// TwinCAT 3 PLC project UiBuilder
// ProgramVersion: 3.1.4026.19
// libraries:
//   Base, * (Photara)
//   Discrete, * (Photara)
//   Motion, * (Photara)
//   Nemo, * (Photara)
//   Tc2_EthernetIP, * (Beckhoff Automation GmbH)
//   Tc2_ProfinetDiag, * (Beckhoff Automation GmbH)
//   Tc2_Standard, * (Beckhoff Automation GmbH)
//   Tc2_System, * (Beckhoff Automation GmbH)
//   Vision, * (Photara)
//   TcUnit, * (www.tcunit.org)
// project tree:
//   DUTs/ ST_HMICommand.TcDUT, ST_HMIConfiguration.TcDUT, ST_HMIComponentAPI.TcDUT, ST_HMIStatus.TcDUT
//   ITFs/ I_HMIBase.TcIO
//   / PlcTask.TcTTO
//   POUs/ FB_HMIBase.TcPOU, MAIN.TcPOU
//   Tests/ FB_ST_HMICommand_Test.TcPOU, FB_ST_HMIComponentAPI_Test.TcPOU, FB_ST_HMIStatus_Test.TcPOU, FB_HMIBase_Test.TcPOU, PRG_TEST.TcPOU

CONFIGURATION UiBuilder
    RESOURCE PLC ON TwinCAT3
        TASK PlcTask(INTERVAL := T#10ms, PRIORITY := 20);
        PROGRAM MAIN WITH PlcTask : MAIN;
    END_RESOURCE
END_CONFIGURATION

// ---- DUTs/ST_HMICommand.TcDUT
TYPE ST_HMICommand :
STRUCT
	Enable	: BOOL;
	Disable	: BOOL;
	Home	: BOOL;
	Reset	: BOOL;
	Stop	: BOOL;
	Trigger	: BOOL;
	Error	: BYTE;
END_STRUCT
END_TYPE

// ---- DUTs/ST_HMIConfiguration.TcDUT
TYPE ST_HMIConfiguration :
STRUCT
	ComponentConfiguration : REFERENCE TO ST_CommandConfiguration;
END_STRUCT
END_TYPE

// ---- DUTs/ST_HMIComponentAPI.TcDUT
TYPE ST_HMIComponentAPI :
STRUCT 
	Done : BOOL;
	Busy : BOOL;
	Error : BOOL;
	ErrorID : BOOL;
	Ready : BOOL;
	Enabled: BOOL;
	Homed: BOOL;
	Moving : BOOL;
END_STRUCT
END_TYPE

// ---- DUTs/ST_HMIStatus.TcDUT
TYPE ST_HMIStatus :
STRUCT
	ComponentStatus : REFERENCE TO ST_ComponentStatus;
	HmiStatus : ST_HmiComponentAPI;
END_STRUCT
END_TYPE

// ---- ITFs/I_HMIBase.TcIO
INTERFACE I_HMIBase EXTENDS	Base.I_BaseCyclic

PROPERTY P_BaseConfiguration : REFERENCE TO ST_BaseConfiguration
GET
END_GET
SET
END_SET
END_PROPERTY

PROPERTY P_BaseStatus : REFERENCE TO ST_BaseStatus
GET
END_GET
SET
END_SET
END_PROPERTY

PROPERTY P_Command : REFERENCE TO P_Command
GET
END_GET
SET
END_SET
END_PROPERTY

END_INTERFACE

// ---- POUs/MAIN.TcPOU
PROGRAM MAIN
VAR
END_VAR

END_PROGRAM

// ---- POUs/FB_HMIBase.TcPOU
FUNCTION_BLOCK FB_HMIBase
VAR
	status : ST_HMIStatus;
	configs : ST_HMIConfiguration;
	cmd : ST_HMICommand;
END_VAR

PROPERTY P_Command : ST_HMICommand
GET
END_GET
SET
END_SET
END_PROPERTY

PROPERTY P_Configuration : ST_HMIConfiguration
GET
END_GET
SET
END_SET
END_PROPERTY

PROPERTY P_Status : ST_HMIStatus
GET
END_GET
SET
END_SET
END_PROPERTY

END_FUNCTION_BLOCK

// ---- Tests/FB_ST_HMICommand_Test.TcPOU
FUNCTION_BLOCK FB_ST_HMICommand_Test EXTENDS TcUnit.FB_TestSuite
VAR_INPUT
END_VAR
VAR_OUTPUT
END_VAR
VAR
	testCommand : ST_HMICommand;
END_VAR

// Test runner - call all test methods
Test_InitialState();
Test_EnableCommand();
Test_DisableCommand();
Test_HomeCommand();
Test_ResetCommand();
Test_StopCommand();
Test_TriggerCommand();
Test_ErrorCode();
Test_MultipleCommands();
Test_ClearCommands();

METHOD Test_InitialState
VAR_INPUT
END_VAR
TEST('Test_InitialState');

// Test that all command flags are initially FALSE
testCommand.Enable := FALSE;
testCommand.Disable := FALSE;
testCommand.Home := FALSE;
testCommand.Reset := FALSE;
testCommand.Stop := FALSE;
testCommand.Trigger := FALSE;
testCommand.Error := 0;

AssertFalse(testCommand.Enable, 'Enable should be FALSE initially');
AssertFalse(testCommand.Disable, 'Disable should be FALSE initially');
AssertFalse(testCommand.Home, 'Home should be FALSE initially');
AssertFalse(testCommand.Reset, 'Reset should be FALSE initially');
AssertFalse(testCommand.Stop, 'Stop should be FALSE initially');
AssertFalse(testCommand.Trigger, 'Trigger should be FALSE initially');
AssertEquals_BYTE(0, testCommand.Error, 'Error should be 0 initially');

TEST_FINISHED();
END_METHOD

METHOD Test_EnableCommand
VAR_INPUT
END_VAR
TEST('Test_EnableCommand');

// Test Enable command can be set
testCommand.Enable := TRUE;
AssertTrue(testCommand.Enable, 'Enable should be TRUE when set');

// Reset
testCommand.Enable := FALSE;
AssertFalse(testCommand.Enable, 'Enable should be FALSE when reset');

TEST_FINISHED();
END_METHOD

METHOD Test_DisableCommand
VAR_INPUT
END_VAR
TEST('Test_DisableCommand');

// Test Disable command can be set
testCommand.Disable := TRUE;
AssertTrue(testCommand.Disable, 'Disable should be TRUE when set');

// Reset
testCommand.Disable := FALSE;
AssertFalse(testCommand.Disable, 'Disable should be FALSE when reset');

TEST_FINISHED();
END_METHOD

METHOD Test_HomeCommand
VAR_INPUT
END_VAR
TEST('Test_HomeCommand');

// Test Home command can be set
testCommand.Home := TRUE;
AssertTrue(testCommand.Home, 'Home should be TRUE when set');

// Reset
testCommand.Home := FALSE;
AssertFalse(testCommand.Home, 'Home should be FALSE when reset');

TEST_FINISHED();
END_METHOD

METHOD Test_ResetCommand
VAR_INPUT
END_VAR
TEST('Test_ResetCommand');

// Test Reset command can be set
testCommand.Reset := TRUE;
AssertTrue(testCommand.Reset, 'Reset should be TRUE when set');

// Reset
testCommand.Reset := FALSE;
AssertFalse(testCommand.Reset, 'Reset should be FALSE when reset');

TEST_FINISHED();
END_METHOD

METHOD Test_StopCommand
VAR_INPUT
END_VAR
TEST('Test_StopCommand');

// Test Stop command can be set
testCommand.Stop := TRUE;
AssertTrue(testCommand.Stop, 'Stop should be TRUE when set');

// Reset
testCommand.Stop := FALSE;
AssertFalse(testCommand.Stop, 'Stop should be FALSE when reset');

TEST_FINISHED();
END_METHOD

METHOD Test_TriggerCommand
VAR_INPUT
END_VAR
TEST('Test_TriggerCommand');

// Test Trigger command can be set
testCommand.Trigger := TRUE;
AssertTrue(testCommand.Trigger, 'Trigger should be TRUE when set');

// Reset
testCommand.Trigger := FALSE;
AssertFalse(testCommand.Trigger, 'Trigger should be FALSE when reset');

TEST_FINISHED();
END_METHOD

METHOD Test_ErrorCode
VAR_INPUT
END_VAR
TEST('Test_ErrorCode');

// Test Error code can be set to various values
testCommand.Error := 0;
AssertEquals_BYTE(0, testCommand.Error, 'Error should be 0');

testCommand.Error := 1;
AssertEquals_BYTE(1, testCommand.Error, 'Error should be 1');

testCommand.Error := 255;
AssertEquals_BYTE(255, testCommand.Error, 'Error should be 255');

testCommand.Error := 128;
AssertEquals_BYTE(128, testCommand.Error, 'Error should be 128');

TEST_FINISHED();
END_METHOD

METHOD Test_MultipleCommands
VAR_INPUT
END_VAR
TEST('Test_MultipleCommands');

// Test multiple commands can be set simultaneously
testCommand.Enable := TRUE;
testCommand.Home := TRUE;
testCommand.Trigger := TRUE;

AssertTrue(testCommand.Enable, 'Enable should be TRUE');
AssertTrue(testCommand.Home, 'Home should be TRUE');
AssertTrue(testCommand.Trigger, 'Trigger should be TRUE');
AssertFalse(testCommand.Disable, 'Disable should remain FALSE');
AssertFalse(testCommand.Stop, 'Stop should remain FALSE');

TEST_FINISHED();
END_METHOD

METHOD Test_ClearCommands
VAR_INPUT
END_VAR
TEST('Test_ClearCommands');

// Set all commands
testCommand.Enable := TRUE;
testCommand.Disable := TRUE;
testCommand.Home := TRUE;
testCommand.Reset := TRUE;
testCommand.Stop := TRUE;
testCommand.Trigger := TRUE;
testCommand.Error := 42;

// Clear all commands
testCommand.Enable := FALSE;
testCommand.Disable := FALSE;
testCommand.Home := FALSE;
testCommand.Reset := FALSE;
testCommand.Stop := FALSE;
testCommand.Trigger := FALSE;
testCommand.Error := 0;

// Verify all are cleared
AssertFalse(testCommand.Enable, 'Enable should be FALSE');
AssertFalse(testCommand.Disable, 'Disable should be FALSE');
AssertFalse(testCommand.Home, 'Home should be FALSE');
AssertFalse(testCommand.Reset, 'Reset should be FALSE');
AssertFalse(testCommand.Stop, 'Stop should be FALSE');
AssertFalse(testCommand.Trigger, 'Trigger should be FALSE');
AssertEquals_BYTE(0, testCommand.Error, 'Error should be 0');

TEST_FINISHED();
END_METHOD

END_FUNCTION_BLOCK

// ---- Tests/FB_ST_HMIComponentAPI_Test.TcPOU
FUNCTION_BLOCK FB_ST_HMIComponentAPI_Test EXTENDS TcUnit.FB_TestSuite
VAR_INPUT
END_VAR
VAR_OUTPUT
END_VAR
VAR
	testAPI : ST_HMIComponentAPI;
END_VAR

// Test runner - call all test methods
Test_InitialState();
Test_DoneFlag();
Test_BusyFlag();
Test_ErrorFlag();
Test_ErrorIDFlag();
Test_ReadyFlag();
Test_EnabledFlag();
Test_HomedFlag();
Test_MovingFlag();
Test_StateTransitions();
Test_ErrorState();
Test_BusyToDone();
Test_AllFlagsSet();
Test_ClearAllFlags();

METHOD Test_InitialState
VAR_INPUT
END_VAR
TEST('Test_InitialState');

// Initialize all flags to FALSE
testAPI.Done := FALSE;
testAPI.Busy := FALSE;
testAPI.Error := FALSE;
testAPI.ErrorID := FALSE;
testAPI.Ready := FALSE;
testAPI.Enabled := FALSE;
testAPI.Homed := FALSE;
testAPI.Moving := FALSE;

// Verify initial state
AssertFalse(testAPI.Done, 'Done should be FALSE initially');
AssertFalse(testAPI.Busy, 'Busy should be FALSE initially');
AssertFalse(testAPI.Error, 'Error should be FALSE initially');
AssertFalse(testAPI.ErrorID, 'ErrorID should be FALSE initially');
AssertFalse(testAPI.Ready, 'Ready should be FALSE initially');
AssertFalse(testAPI.Enabled, 'Enabled should be FALSE initially');
AssertFalse(testAPI.Homed, 'Homed should be FALSE initially');
AssertFalse(testAPI.Moving, 'Moving should be FALSE initially');

TEST_FINISHED();
END_METHOD

METHOD Test_DoneFlag
VAR_INPUT
END_VAR
TEST('Test_DoneFlag');

// Test Done flag can be set
testAPI.Done := TRUE;
AssertTrue(testAPI.Done, 'Done should be TRUE when set');

// Reset
testAPI.Done := FALSE;
AssertFalse(testAPI.Done, 'Done should be FALSE when reset');

TEST_FINISHED();
END_METHOD

METHOD Test_BusyFlag
VAR_INPUT
END_VAR
TEST('Test_BusyFlag');

// Test Busy flag can be set
testAPI.Busy := TRUE;
AssertTrue(testAPI.Busy, 'Busy should be TRUE when set');

// Reset
testAPI.Busy := FALSE;
AssertFalse(testAPI.Busy, 'Busy should be FALSE when reset');

TEST_FINISHED();
END_METHOD

METHOD Test_ErrorFlag
VAR_INPUT
END_VAR
TEST('Test_ErrorFlag');

// Test Error flag can be set
testAPI.Error := TRUE;
AssertTrue(testAPI.Error, 'Error should be TRUE when set');

// Reset
testAPI.Error := FALSE;
AssertFalse(testAPI.Error, 'Error should be FALSE when reset');

TEST_FINISHED();
END_METHOD

METHOD Test_ErrorIDFlag
VAR_INPUT
END_VAR
TEST('Test_ErrorIDFlag');

// Test ErrorID flag can be set
testAPI.ErrorID := TRUE;
AssertTrue(testAPI.ErrorID, 'ErrorID should be TRUE when set');

// Reset
testAPI.ErrorID := FALSE;
AssertFalse(testAPI.ErrorID, 'ErrorID should be FALSE when reset');

TEST_FINISHED();
END_METHOD

METHOD Test_ReadyFlag
VAR_INPUT
END_VAR
TEST('Test_ReadyFlag');

// Test Ready flag can be set
testAPI.Ready := TRUE;
AssertTrue(testAPI.Ready, 'Ready should be TRUE when set');

// Reset
testAPI.Ready := FALSE;
AssertFalse(testAPI.Ready, 'Ready should be FALSE when reset');

TEST_FINISHED();
END_METHOD

METHOD Test_EnabledFlag
VAR_INPUT
END_VAR
TEST('Test_EnabledFlag');

// Test Enabled flag can be set
testAPI.Enabled := TRUE;
AssertTrue(testAPI.Enabled, 'Enabled should be TRUE when set');

// Reset
testAPI.Enabled := FALSE;
AssertFalse(testAPI.Enabled, 'Enabled should be FALSE when reset');

TEST_FINISHED();
END_METHOD

METHOD Test_HomedFlag
VAR_INPUT
END_VAR
TEST('Test_HomedFlag');

// Test Homed flag can be set
testAPI.Homed := TRUE;
AssertTrue(testAPI.Homed, 'Homed should be TRUE when set');

// Reset
testAPI.Homed := FALSE;
AssertFalse(testAPI.Homed, 'Homed should be FALSE when reset');

TEST_FINISHED();
END_METHOD

METHOD Test_MovingFlag
VAR_INPUT
END_VAR
TEST('Test_MovingFlag');

// Test Moving flag can be set
testAPI.Moving := TRUE;
AssertTrue(testAPI.Moving, 'Moving should be TRUE when set');

// Reset
testAPI.Moving := FALSE;
AssertFalse(testAPI.Moving, 'Moving should be FALSE when reset');

TEST_FINISHED();
END_METHOD

METHOD Test_StateTransitions
VAR_INPUT
END_VAR
TEST('Test_StateTransitions');

// Simulate typical state transition: Ready -> Busy -> Done
testAPI.Ready := TRUE;
AssertTrue(testAPI.Ready, 'Should be Ready initially');
AssertFalse(testAPI.Busy, 'Should not be Busy initially');
AssertFalse(testAPI.Done, 'Should not be Done initially');

// Transition to Busy
testAPI.Busy := TRUE;
testAPI.Ready := FALSE;
AssertFalse(testAPI.Ready, 'Should not be Ready when Busy');
AssertTrue(testAPI.Busy, 'Should be Busy');
AssertFalse(testAPI.Done, 'Should not be Done while Busy');

// Transition to Done
testAPI.Done := TRUE;
testAPI.Busy := FALSE;
AssertFalse(testAPI.Busy, 'Should not be Busy when Done');
AssertTrue(testAPI.Done, 'Should be Done');

TEST_FINISHED();
END_METHOD

METHOD Test_ErrorState
VAR_INPUT
END_VAR
TEST('Test_ErrorState');

// Simulate error condition
testAPI.Error := TRUE;
testAPI.ErrorID := TRUE;
testAPI.Busy := FALSE;
testAPI.Done := FALSE;

AssertTrue(testAPI.Error, 'Error should be TRUE');
AssertTrue(testAPI.ErrorID, 'ErrorID should be TRUE');
AssertFalse(testAPI.Done, 'Done should be FALSE in error state');
AssertFalse(testAPI.Busy, 'Busy should be FALSE in error state');

TEST_FINISHED();
END_METHOD

METHOD Test_BusyToDone
VAR_INPUT
END_VAR
TEST('Test_BusyToDone');

// Test transition from Busy to Done (should be mutually exclusive)
testAPI.Busy := TRUE;
testAPI.Done := FALSE;
AssertTrue(testAPI.Busy, 'Should be Busy');
AssertFalse(testAPI.Done, 'Done should be FALSE when Busy');

// Complete operation
testAPI.Busy := FALSE;
testAPI.Done := TRUE;
AssertFalse(testAPI.Busy, 'Busy should be FALSE when Done');
AssertTrue(testAPI.Done, 'Should be Done');

TEST_FINISHED();
END_METHOD

METHOD Test_AllFlagsSet
VAR_INPUT
END_VAR
TEST('Test_AllFlagsSet');

// Test that all flags can be set simultaneously (though not typical in practice)
testAPI.Done := TRUE;
testAPI.Busy := TRUE;
testAPI.Error := TRUE;
testAPI.ErrorID := TRUE;
testAPI.Ready := TRUE;
testAPI.Enabled := TRUE;
testAPI.Homed := TRUE;
testAPI.Moving := TRUE;

AssertTrue(testAPI.Done, 'Done should be TRUE');
AssertTrue(testAPI.Busy, 'Busy should be TRUE');
AssertTrue(testAPI.Error, 'Error should be TRUE');
AssertTrue(testAPI.ErrorID, 'ErrorID should be TRUE');
AssertTrue(testAPI.Ready, 'Ready should be TRUE');
AssertTrue(testAPI.Enabled, 'Enabled should be TRUE');
AssertTrue(testAPI.Homed, 'Homed should be TRUE');
AssertTrue(testAPI.Moving, 'Moving should be TRUE');

TEST_FINISHED();
END_METHOD

METHOD Test_ClearAllFlags
VAR_INPUT
END_VAR
TEST('Test_ClearAllFlags');

// Set all flags
testAPI.Done := TRUE;
testAPI.Busy := TRUE;
testAPI.Error := TRUE;
testAPI.ErrorID := TRUE;
testAPI.Ready := TRUE;
testAPI.Enabled := TRUE;
testAPI.Homed := TRUE;
testAPI.Moving := TRUE;

// Clear all flags
testAPI.Done := FALSE;
testAPI.Busy := FALSE;
testAPI.Error := FALSE;
testAPI.ErrorID := FALSE;
testAPI.Ready := FALSE;
testAPI.Enabled := FALSE;
testAPI.Homed := FALSE;
testAPI.Moving := FALSE;

// Verify all are cleared
AssertFalse(testAPI.Done, 'Done should be FALSE');
AssertFalse(testAPI.Busy, 'Busy should be FALSE');
AssertFalse(testAPI.Error, 'Error should be FALSE');
AssertFalse(testAPI.ErrorID, 'ErrorID should be FALSE');
AssertFalse(testAPI.Ready, 'Ready should be FALSE');
AssertFalse(testAPI.Enabled, 'Enabled should be FALSE');
AssertFalse(testAPI.Homed, 'Homed should be FALSE');
AssertFalse(testAPI.Moving, 'Moving should be FALSE');

TEST_FINISHED();
END_METHOD

END_FUNCTION_BLOCK

// ---- Tests/FB_ST_HMIStatus_Test.TcPOU
FUNCTION_BLOCK FB_ST_HMIStatus_Test EXTENDS TcUnit.FB_TestSuite
VAR_INPUT
END_VAR
VAR_OUTPUT
END_VAR
VAR
	testStatus : ST_HMIStatus;
END_VAR

// Test runner - call all test methods
Test_InitialState();
Test_HmiStatusAccess();
Test_HmiStatusFlags();
Test_HmiStatusStateTransitions();

METHOD Test_InitialState
VAR_INPUT
END_VAR
TEST('Test_InitialState');

// Initialize HmiStatus structure
testStatus.HmiStatus.Done := FALSE;
testStatus.HmiStatus.Busy := FALSE;
testStatus.HmiStatus.Error := FALSE;
testStatus.HmiStatus.ErrorID := FALSE;
testStatus.HmiStatus.Ready := FALSE;
testStatus.HmiStatus.Enabled := FALSE;
testStatus.HmiStatus.Homed := FALSE;
testStatus.HmiStatus.Moving := FALSE;

// Verify initial state of HmiStatus member
AssertFalse(testStatus.HmiStatus.Done, 'HmiStatus.Done should be FALSE initially');
AssertFalse(testStatus.HmiStatus.Busy, 'HmiStatus.Busy should be FALSE initially');
AssertFalse(testStatus.HmiStatus.Error, 'HmiStatus.Error should be FALSE initially');
AssertFalse(testStatus.HmiStatus.ErrorID, 'HmiStatus.ErrorID should be FALSE initially');
AssertFalse(testStatus.HmiStatus.Ready, 'HmiStatus.Ready should be FALSE initially');
AssertFalse(testStatus.HmiStatus.Enabled, 'HmiStatus.Enabled should be FALSE initially');
AssertFalse(testStatus.HmiStatus.Homed, 'HmiStatus.Homed should be FALSE initially');
AssertFalse(testStatus.HmiStatus.Moving, 'HmiStatus.Moving should be FALSE initially');

TEST_FINISHED();
END_METHOD

METHOD Test_HmiStatusAccess
VAR_INPUT
END_VAR
TEST('Test_HmiStatusAccess');

// Test that HmiStatus member can be accessed and modified
testStatus.HmiStatus.Ready := TRUE;
AssertTrue(testStatus.HmiStatus.Ready, 'HmiStatus.Ready should be accessible and settable');

testStatus.HmiStatus.Enabled := TRUE;
AssertTrue(testStatus.HmiStatus.Enabled, 'HmiStatus.Enabled should be accessible and settable');

testStatus.HmiStatus.Homed := TRUE;
AssertTrue(testStatus.HmiStatus.Homed, 'HmiStatus.Homed should be accessible and settable');

TEST_FINISHED();
END_METHOD

METHOD Test_HmiStatusFlags
VAR_INPUT
END_VAR
TEST('Test_HmiStatusFlags');

// Test all HmiStatus flags can be set independently
testStatus.HmiStatus.Done := TRUE;
testStatus.HmiStatus.Busy := FALSE;
testStatus.HmiStatus.Error := FALSE;

AssertTrue(testStatus.HmiStatus.Done, 'Done flag should be TRUE');
AssertFalse(testStatus.HmiStatus.Busy, 'Busy flag should be FALSE');
AssertFalse(testStatus.HmiStatus.Error, 'Error flag should be FALSE');

// Change state
testStatus.HmiStatus.Done := FALSE;
testStatus.HmiStatus.Busy := TRUE;

AssertFalse(testStatus.HmiStatus.Done, 'Done flag should be FALSE');
AssertTrue(testStatus.HmiStatus.Busy, 'Busy flag should be TRUE');

TEST_FINISHED();
END_METHOD

METHOD Test_HmiStatusStateTransitions
VAR_INPUT
END_VAR
TEST('Test_HmiStatusStateTransitions');

// Test typical state machine transitions through HmiStatus
// Initial state: Ready
testStatus.HmiStatus.Ready := TRUE;
testStatus.HmiStatus.Enabled := FALSE;
testStatus.HmiStatus.Busy := FALSE;
testStatus.HmiStatus.Done := FALSE;

AssertTrue(testStatus.HmiStatus.Ready, 'Should be Ready initially');

// Enabled state
testStatus.HmiStatus.Enabled := TRUE;
AssertTrue(testStatus.HmiStatus.Enabled, 'Should be Enabled');
AssertTrue(testStatus.HmiStatus.Ready, 'Should remain Ready when Enabled');

// Busy executing
testStatus.HmiStatus.Busy := TRUE;
testStatus.HmiStatus.Done := FALSE;
AssertTrue(testStatus.HmiStatus.Busy, 'Should be Busy');
AssertFalse(testStatus.HmiStatus.Done, 'Should not be Done while Busy');

// Completed
testStatus.HmiStatus.Busy := FALSE;
testStatus.HmiStatus.Done := TRUE;
AssertFalse(testStatus.HmiStatus.Busy, 'Should not be Busy when Done');
AssertTrue(testStatus.HmiStatus.Done, 'Should be Done');

TEST_FINISHED();
END_METHOD

END_FUNCTION_BLOCK

// ---- Tests/FB_HMIBase_Test.TcPOU
FUNCTION_BLOCK FB_HMIBase_Test EXTENDS TcUnit.FB_TestSuite
VAR_INPUT
END_VAR
VAR_OUTPUT
END_VAR
VAR
	testFB : FB_HMIBase;
	testCommand : ST_HMICommand;
	testConfig : ST_HMIConfiguration;
	testStatus : ST_HMIStatus;
END_VAR

// Test runner - call all test methods
Test_FunctionBlockInstantiation();
Test_CommandProperty();how 
Test_ConfigurationProperty();
Test_StatusProperty();
Test_CommandPropertyReadWrite();
Test_StatusPropertyRead();
Test_ConfigurationPropertyReadWrite();

METHOD Test_CommandProperty
VAR_INPUT
END_VAR
VAR
	retrievedCommand : ST_HMICommand;
END_VAR
TEST('Test_CommandProperty');

// Test P_Command property
// Note: This test assumes property implementation will be added
// Once properties are implemented, this will verify getter/setter behavior

// Set up test command
testCommand.Enable := TRUE;
testCommand.Home := TRUE;
testCommand.Reset := FALSE;

// Note: When properties are implemented, uncomment:
// testFB.P_Command := testCommand;
// retrievedCommand := testFB.P_Command;
// AssertTrue(retrievedCommand.Enable, 'Command.Enable should be TRUE');
// AssertTrue(retrievedCommand.Home, 'Command.Home should be TRUE');
// AssertFalse(retrievedCommand.Reset, 'Command.Reset should be FALSE');

// For now, just verify the structure works
AssertTrue(testCommand.Enable, 'Test command Enable flag works');

TEST_FINISHED();
END_METHOD

METHOD Test_CommandPropertyReadWrite
VAR_INPUT
END_VAR
VAR
	writeCommand : ST_HMICommand;
	readCommand : ST_HMICommand;
END_VAR
TEST('Test_CommandPropertyReadWrite');

// Prepare test data
writeCommand.Enable := TRUE;
writeCommand.Disable := FALSE;
writeCommand.Home := TRUE;
writeCommand.Reset := FALSE;
writeCommand.Stop := FALSE;
writeCommand.Trigger := TRUE;
writeCommand.Error := 42;

// When property implementation is complete, this will test:
// 1. Write via property setter
// testFB.P_Command := writeCommand;

// 2. Read via property getter
// readCommand := testFB.P_Command;

// 3. Verify data integrity
// AssertTrue(readCommand.Enable, 'Enable should match written value');
// AssertFalse(readCommand.Disable, 'Disable should match written value');
// AssertTrue(readCommand.Home, 'Home should match written value');
// AssertTrue(readCommand.Trigger, 'Trigger should match written value');
// AssertEquals_BYTE(42, readCommand.Error, 'Error code should match written value');

// Placeholder verification
AssertTrue(writeCommand.Enable, 'Write command prepared correctly');

TEST_FINISHED();
END_METHOD

METHOD Test_ConfigurationProperty
VAR_INPUT
END_VAR
VAR
	retrievedConfig : ST_HMIConfiguration;
END_VAR
TEST('Test_ConfigurationProperty');

// Test P_Configuration property
// Note: This test assumes property implementation will be added

// Set up test configuration
// testConfig is ready to use once properties are implemented

// Note: When properties are implemented, uncomment:
// testFB.P_Configuration := testConfig;
// retrievedConfig := testFB.P_Configuration;

// For now, verify the structure exists
AssertTrue(TRUE, 'Configuration structure is defined');

TEST_FINISHED();
END_METHOD

METHOD Test_ConfigurationPropertyReadWrite
VAR_INPUT
END_VAR
VAR
	writeConfig : ST_HMIConfiguration;
	readConfig : ST_HMIConfiguration;
END_VAR
TEST('Test_ConfigurationPropertyReadWrite');

// Test configuration property read/write
// Configurations are typically set once and read multiple times

// When property implementation is complete:
// testFB.P_Configuration := writeConfig;
// readConfig := testFB.P_Configuration;

// Verify configuration was stored correctly
// (Will need actual configuration values once ST_CommandConfiguration is defined)

// Placeholder verification
AssertTrue(TRUE, 'Configuration property structure is ready for implementation');

TEST_FINISHED();
END_METHOD

METHOD Test_FunctionBlockInstantiation
VAR_INPUT
END_VAR
TEST('Test_FunctionBlockInstantiation');

// Test that FB_HMIBase can be instantiated
// The mere fact that testFB exists and this test runs proves instantiation works
AssertTrue(TRUE, 'FB_HMIBase should be instantiable');

TEST_FINISHED();
END_METHOD

METHOD Test_StatusProperty
VAR_INPUT
END_VAR
VAR
	retrievedStatus : ST_HMIStatus;
END_VAR
TEST('Test_StatusProperty');

// Test P_Status property
// Note: This test assumes property implementation will be added

// Set up test status
testStatus.HmiStatus.Ready := TRUE;
testStatus.HmiStatus.Enabled := TRUE;

// Note: When properties are implemented, uncomment:
// testFB.P_Status := testStatus;
// retrievedStatus := testFB.P_Status;
// AssertTrue(retrievedStatus.HmiStatus.Ready, 'Status.HmiStatus.Ready should be TRUE');
// AssertTrue(retrievedStatus.HmiStatus.Enabled, 'Status.HmiStatus.Enabled should be TRUE');

// For now, verify the structure works
AssertTrue(testStatus.HmiStatus.Ready, 'Test status Ready flag works');

TEST_FINISHED();
END_METHOD

METHOD Test_StatusPropertyRead
VAR_INPUT
END_VAR
VAR
	readStatus : ST_HMIStatus;
END_VAR
TEST('Test_StatusPropertyRead');

// Typically status is read-only from external perspective
// This test verifies status can be read via property

// When property implementation is complete:
// readStatus := testFB.P_Status;

// Verify status flags can be read
// AssertFalse(readStatus.HmiStatus.Error, 'Should be able to read Error flag');
// AssertFalse(readStatus.HmiStatus.Busy, 'Should be able to read Busy flag');

// Placeholder verification
AssertTrue(TRUE, 'Status property structure is ready for implementation');

TEST_FINISHED();
END_METHOD

END_FUNCTION_BLOCK

// ---- Tests/PRG_TEST.TcPOU
PROGRAM PRG_TEST
VAR
	// Test suite instances
	fbCommandTest : FB_ST_HMICommand_Test;
	fbComponentAPITest : FB_ST_HMIComponentAPI_Test;
	fbStatusTest : FB_ST_HMIStatus_Test;
	fbHMIBaseTest : FB_HMIBase_Test;
END_VAR

// ============================================================================
// UiBuilder Library Test Suite
// ============================================================================
// This program runs all unit tests for the UiBuilder library using TcUnit
// framework. Call this program from your main task to execute tests.
//
// Test Coverage:
// - ST_HMICommand data type tests
// - ST_HMIComponentAPI data type tests
// - ST_HMIStatus data type tests
// - FB_HMIBase function block tests
//
// Usage:
// 1. Add PRG_TEST to your PlcTask or call from MAIN
// 2. Build and download the project
// 3. Run the PLC
// 4. Check TcUnit results in the output window
// ============================================================================

// Execute all test suites
// TcUnit automatically collects and reports results through FB_TestSuite base class
fbCommandTest();
fbComponentAPITest();
fbStatusTest();
fbHMIBaseTest();

END_PROGRAM
